// Mitsubishi GX Works2 project: BookEX6_38 Display   PLC: Q13UDV

// global labels: Global
VAR_GLOBAL
  bVar0 AT M5000 : BOOL;
  abArray0 AT M5010 : ARRAY [0..49] OF BOOL;
  sStr0 AT D5000 : STRING[199];
  sStr1 AT D5100 : STRING[199];
  sStr2 AT D5200 : STRING[199];
  sStr3 AT D5300 : STRING[199];
  sStr4 AT D5400 : STRING[199];
  sStr5 AT D5500 : STRING[199];
  sStr6 AT D5600 : STRING[199];
  sStr7 AT D5700 : STRING[199];
  sStr8 AT D5800 : STRING[199];
  sStr9 AT D5900 : STRING[199];
  iVar0 AT D4500 : INT;
  iVar1 AT D4501 : INT;
  iVar2 AT D4502 : INT;
  iVar3 AT D4503 : INT;
  iVar4 AT D4504 : INT;
  iVar5 AT D4505 : INT;
  iVar6 AT D4506 : INT;
  iVar7 AT D4507 : INT;
  iVar8 AT D4508 : INT;
  iVar9 AT D4509 : INT;
  dVar0 AT D4510 : DINT;
  dVar1 AT D4512 : DINT;
  dVar2 AT D4514 : DINT;
  dVar3 AT D4516 : DINT;
  dVar4 AT D4518 : DINT;
  dVar5 AT D4520 : DINT;
  dVar6 AT D4522 : DINT;
  dVar7 AT D4524 : DINT;
  dVar8 AT D4526 : DINT;
  dVar9 AT D4528 : DINT;
  wVar0 AT D4530 : WORD;
  wVar1 AT D4531 : WORD;
  wVar2 AT D4532 : WORD;
  wVar3 AT D4533 : WORD;
  wVar4 AT D4534 : WORD;
  wVar5 AT D4535 : WORD;
  wVar6 AT D4536 : WORD;
  wVar7 AT D4537 : WORD;
  wVar8 AT D4538 : WORD;
  wVar9 AT D4539 : WORD;
  dwVar0 AT D4540 : DWORD;
  dwVar1 AT D4542 : DWORD;
  dwVar2 AT D4544 : DWORD;
  dwVar3 AT D4546 : DWORD;
  dwVar4 AT D4548 : DWORD;
  dwVar5 AT D4550 : DWORD;
  dwVar6 AT D4552 : DWORD;
  dwVar7 AT D4554 : DWORD;
  dwVar8 AT D4556 : DWORD;
  dwVar9 AT D4558 : DWORD;
  fsVar0 AT D4560 : REAL;
  fsVar1 AT D4562 : REAL;
  fsVar2 AT D4564 : REAL;
  fsVar3 AT D4566 : REAL;
  fsVar4 AT D4568 : REAL;
  fsVar5 AT D4570 : REAL;
  fsVar6 AT D4572 : REAL;
  fsVar7 AT D4574 : REAL;
  fsVar8 AT D4576 : REAL;
  fsVar9 AT D4578 : REAL;
  fdVar0 AT D4580 : LREAL;
  tTime0 AT D4620 : TIME;
  tTime1 AT D4622 : TIME;
  tTime2 AT D4624 : TIME;
  tTime3 AT D4626 : TIME;
  tTime4 AT D4628 : TIME;
  tTime5 AT D4630 : TIME;
  tTime6 AT D4632 : TIME;
  tTime7 AT D4634 : TIME;
  tTime8 AT D4636 : TIME;
  tTime9 AT D4638 : TIME;
  tTime10 AT D4640 : TIME;
  bVar1 AT M5001 : BOOL;
  bVar2 AT M5002 : BOOL;
  bVar3 AT M5003 : BOOL;
  bVar4 AT M5004 : BOOL;
  bVar5 AT M5005 : BOOL;
  bVar6 AT M5006 : BOOL;
  bVar7 AT M5007 : BOOL;
  bVar8 AT M5008 : BOOL;
  bVar9 AT M5009 : BOOL;
  abArray1 AT M5060 : ARRAY [0..49] OF BOOL;
  abArray2 AT M5110 : ARRAY [0..49] OF BOOL;
  abArray3 AT M5160 : ARRAY [0..49] OF BOOL;
  abArray4 AT M5210 : ARRAY [0..49] OF BOOL;
  abArray5 AT M5260 : ARRAY [0..49] OF BOOL;
  abArray6 AT M5310 : ARRAY [0..49] OF BOOL;
  abArray7 AT M5360 : ARRAY [0..49] OF BOOL;
  abArray8 AT M5410 : ARRAY [0..49] OF BOOL;
  abArray9 AT M5460 : ARRAY [0..49] OF BOOL;
  fdVar1 AT D4584 : LREAL;
  fdVar2 AT D4588 : LREAL;
  fdVar3 AT D4592 : LREAL;
  fdVar4 AT D4596 : LREAL;
  fdVar5 AT D4600 : LREAL;
  fdVar6 AT D4604 : LREAL;
  fdVar7 AT D4608 : LREAL;
  fdVar8 AT D4612 : LREAL;
  fdVar9 AT D4616 : LREAL;
  afsPen0 AT D2000 : ARRAY [0..499] OF REAL;
  afsPen1 AT D3000 : ARRAY [0..499] OF REAL;
  adwD10 AT D10 : ARRAY [0..9] OF DWORD;
  awD10 AT D10 : ARRAY [0..19] OF WORD;
  BackF AT D100 : ARRAY [0..3,0..99] OF INT;
  abM10 AT M10 : ARRAY [0..19] OF BOOL;
END_VAR
// user libraries (not included): HMI

FUNCTION_BLOCK Backup
VAR_INPUT
  b_EN : BOOL;
  i_Start : INT;
  i_End : INT;
  b_Bit : BOOL;
END_VAR
VAR_OUTPUT
  b_ENO : BOOL;
END_VAR
VAR
  ix : INT;
  iy : INT;
END_VAR
;
IF NOT LDP(TRUE, b_EN) THEN
	b_ENO := FALSE;
	RETURN;
END_IF;
b_ENO := TRUE;
FOR ix := 3 TO 1 BY -1 DO
	FOR iy := i_Start TO i_End DO
		BackF[ix, iy] := BackF[ix-1, iy];
	END_FOR;
END_FOR;
FOR iy := i_Start TO i_End DO
 	Z0 := iy;
	BackF[0, iy] := SD0Z0;  
END_FOR;
BackF[0, i_End+1] := BOOL_TO_INT(b_Bit);
END_FUNCTION_BLOCK

FUNCTION_BLOCK sysCpuLed
VAR_OUTPUT
  b_LedMode : BOOL;
  b_LedRun : BOOL;
  b_LedError : BOOL;
  b_LedUser : BOOL;
  b_LedBatt : BOOL;
  b_LedBoot : BOOL;
  i_PLCErrorCode : INT;
END_VAR
VAR
  wLED : WORD;
END_VAR
;
wLED := SD201;
b_LedMode := NOT ((wLED AND HC000) = 0);
b_LedRun := NOT ((wLED AND H0003) = 0);
b_LedError := NOT ((wLED AND H000C) = 0);
b_LedUser := NOT ((wLED AND H0030) = 0);
b_LedBatt := NOT ((wLED AND H00C0) = 0);
b_LedBoot := NOT ((wLED AND H0300) = 0);
(* PLC Error Code *)
i_PLCErrorCode := SD0;
END_FUNCTION_BLOCK

PROGRAM ExCPU
VAR
  sysCpuLed_1 : sysCpuLed;
END_VAR
(* structured ladder/FBD written out as ST: instructions are called as NAME(EN, inputs, outputs); _pN, _eN, _tN stand for wires *)
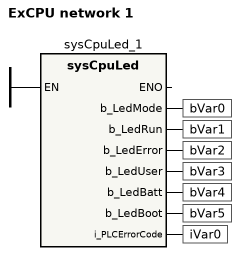
(* network 1 *)
sysCpuLed_1(EN := TRUE, b_LedMode => bVar0, b_LedRun => bVar1, b_LedError => bVar2, b_LedUser => bVar3, b_LedBatt => bVar4, b_LedBoot => bVar5, i_PLCErrorCode => iVar0);
END_PROGRAM

PROGRAM ExF
VAR
  Backup_1 : Backup;
END_VAR
(* structured ladder/FBD written out as ST: instructions are called as NAME(EN, inputs, outputs); _pN, _eN, _tN stand for wires *)
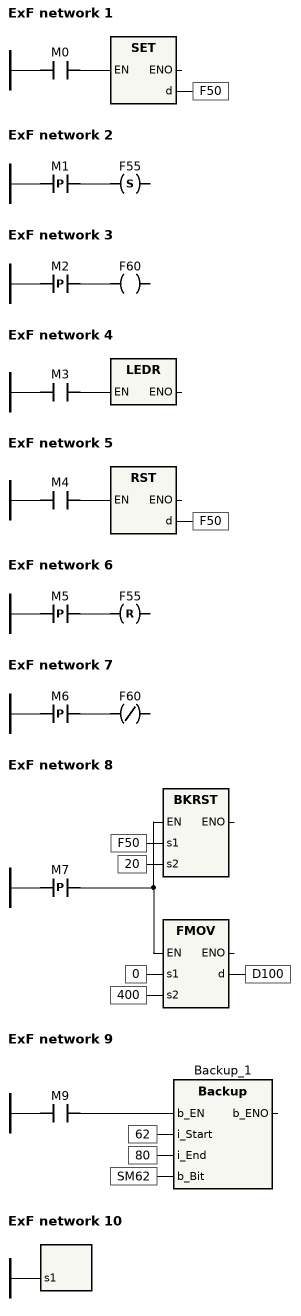
(* network 1 *)
SET(M0, F50);
(* network 2 *)
SET(LDP(TRUE, M1), F55);
(* network 3 *)
F60 := LDP(TRUE, M2);
(* network 4 *)
LEDR(M3);
(* network 5 *)
RST(M4, F50);
(* network 6 *)
RST(LDP(TRUE, M5), F55);
(* network 7 *)
F60 := NOT LDP(TRUE, M6);
(* network 8 *)
_p1 := LDP(TRUE, M7);
BKRST(_p1, F50, 20);
FMOV(_p1, 0, 400, D100);
(* network 9 *)
Backup_1(b_EN := M9, i_Start := 62, i_End := 80, b_Bit := SM62);
(* network 10 *)
(* element kind 10  <- TRUE *)
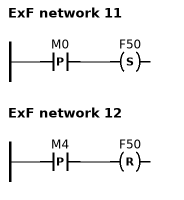
(* network 11 *)
SET(LDP(TRUE, M0), F50);
(* network 12 *)
RST(LDP(TRUE, M4), F50);
END_PROGRAM
